ABB RobotStudio station: Tp2_20201215-221945.rsstn

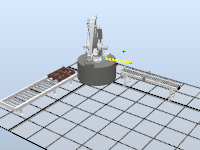
Station Tp2 (saved by RobotStudio 20.2.9116.0)
Controller Controlador1
  mechanical unit ROB_1: IRB660_180_315__01_2, 6 joints, base frame (0, 0, 1000) mm
Layout (positions relative to the parent item):
  - transporteCajas [part, from Equipment\Conveyor Guide 400.rslib] at (0, 1500, 0) mm, rotated rx 0 ry 0 rz 90 deg
  - Euro Pallet [graphiccomponentgroup, from Equipment\Euro Pallet.rslib] at (1000, -1425, 435) mm
    - Body 1 [part, from Equipment\Euro Pallet.rslib]
  - transportePallets [part, from Equipment\Conveyor 950 4000 h2.rslib] at (1000, -1500, 0) mm
  - IRB660_180_315__01_2 [mechanism, from Robots\IRB660_180_315__01.rslib] at (0, 0, 1000) mm; joint values [0.4389, 0.3282, 0.9586, 1.2589] (rad or m)
  - ventosa_tool [mechanism] at (1582.67, 743.05, 1659.86) mm, rotated rx 180 ry 0 rz 133.02 deg
      TCP ventosa_tool at (0, 0, 200) mm
      links: ventosa
  - pedestal [part]
  - fuenteBloques [smart component] at (-200, 1500, 770) mm
      signals: DI agarrar, DO cajaLista
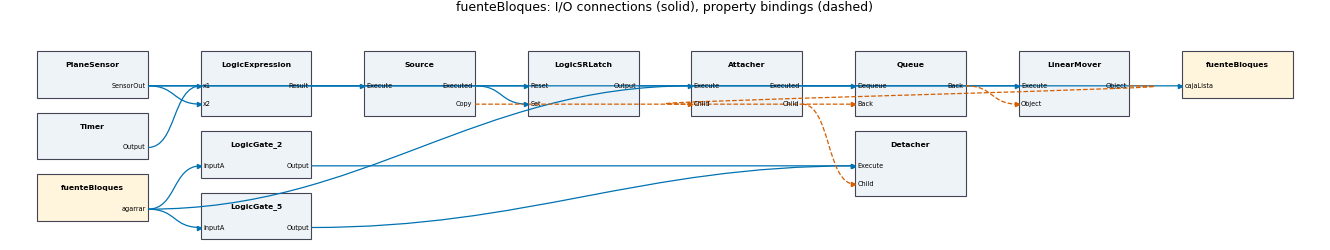
      connections:
        LogicSRLatch.Output -> LinearMover.Execute
        PlaneSensor.SensorOut -> LogicSRLatch.Reset
        Timer.Output -> LogicExpression.x1
        PlaneSensor.SensorOut -> LogicExpression.x2
        LogicExpression.Result -> Source.Execute
        Source.Executed -> LogicSRLatch.Set
        LogicGate_2.Output -> Detacher.Execute
        fuenteBloques.agarrar -> Attacher.Execute
        fuenteBloques.agarrar -> LogicGate_2.InputA
        PlaneSensor.SensorOut -> fuenteBloques.cajaLista
        Attacher.Executed -> Queue.Dequeue
        LogicGate_5.Output -> Detacher.Execute
        fuenteBloques.agarrar -> LogicGate_5.InputA
        Queue.Back => LinearMover.Object
        Source.Copy => Queue.Back
        LinearMover.Object => Attacher.Child
        Attacher.Child => Detacher.Child
    - Source [smart component, from Components\Source.rslib]
        properties: Source=caja; Copy=(none); Parent=(none); Position=[0 2.5 0]; Orientation=[0 0 0]; Transient=true; PhysicsBehavior=0
    - Timer [smart component, from Components\Timer.rslib]
        properties: StartTime=0; Interval=5; Repeat=true; CurrentTime=38.328
    - LinearMover [smart component, from Components\LinearMover.rslib]
        properties: Object=(none); Direction=[0 2.5 0]; Speed=-0.8; Reference=Local; ReferenceObject=fuenteBloques
    - PlaneSensor [smart component, from Components\PlaneSensor.rslib]
        properties: Origin=[-0.1 0.00100000000000011 0]; Axis1=[0 0 0.2]; Axis2=[0.2 0 0]; SensedPart=(none)
      - _sensorPart_ [part]
    - Queue [smart component, from Components\Queue.rslib]
        properties: Back=(none); Front=(none); Queue={b09acd23-45e5-4a9e-9d6f-6607265ff7c3};{23adc33f-3970-47e8-9e1c-f26a8dcf2bdc};{0d33cf10-6771-4310-8fb9-7d79b60af7e9};{83ef1169-329e-4ff4-9302-6302975186d9};{5ada7f3c-b0af-4a10-911f-6c2619dd6db8};{32b629fe-78aa-4961-aeab-383a7d5acd1b};{d9da9d26-80fb-4a26-bfbf-3b7bce0f61f2};{004fb7e2-83f2-4b9c-9668-500ebdcf4198};{63642d38-358b-4db6-ae17-5b4735758ac7};{fa627562-ab66-4e6f-ae79-46c97ebec96c};{c4f368e0-0d9a-4f43-8682-49ac6b133d0c};{43fd2dfd-2b72-4e17-8785-66f02cec94a6};{360d026e-603c-48f5-a2c0-6adaf5a54dd8};{faa924fc-b9a8-4cba-b3be-a1ab497ef86c};{72ea9125-d9f7-4887-b297-381c21b0fe64};{75f844bc-79ed-41e2-8179-ecb24b3a711f};{b9ae99bd-1fa5-4485-ae31-d081ce819117};{bdc3d345-f343-47d8-ada2-183b74e07857};{f98fed9e-0c76-4123-ac69-ce9101c203d3};{b8a068de-0981-4d01-b020-79f46d4aa61e};{6264e575-37ac-44c5-a35d-08152de0ecc4};{b9b05183-98bc-44b7-a44f-bd382026ea01};{e5950468-f040-4ced-9b2d-1f0ddcc9779f};{6daa5a7e-70c7-4fac-8eb8-a3f139030eec};{8209126b-952b-4f15-910a-db478de95a8e};{d94d3c0f-845f-4a91-8578-673738cefad5};{24218f6e-c39a-41e5-a039-2996c01a528f};{42922201-3d4c-4c3c-953c-a9a2c1819590};{11ce3d81-70fa-4fc5-817a-ad43dfd073f9};{d61a1e4e-17c4-421e-8ebd-c30096442b35};{77fdfff2-3eeb-40ed-8391-02d9a381d090};{a548ec3f-cf89-447b-a6c2-8c75641f384b};{21203246-2e5c-4335-a9cf-3c7fcd6009a5};{d9f34a10-d6ad-42c0-8e94-537fdd9e4098};{7434c9e7-4537-4421-8e6c-89bc8283500f};{b2407604-a6d2-40e8-b86b-a185e6f9dabb};{cfdb3468-085d-4a52-9af9-b93c9a7d77cb};{67c8250b-e61e-4164-96c4-8534bc7f99f1};{f8f70fdc-2725-4632-89b5-dc566ac6d74b};{9039b24f-4283-43ad-8f64-d17edb5e158d};{16ad2cc8-d29d-4a04-b806-8d5c79e89c70};{98e4d611-1296-4b4a-afc7-87a9f4683c65};{ea268e05-d762-4d6c-aedb-f9d60f45238b};{23698e1b-885b-404a-990f-58416227340d};{20caccea-1c23-41cc-8a6c-5124b1a7f711}; NumberOfObjects=1
    - caja [part]
    - LogicSRLatch [smart component, from Components\LogicSRLatch.rslib]
    - LogicExpression [smart component, from Components\LogicExpression.rslib]
        properties: Expression=x1 AND NOT x2
    - Attacher [smart component, from Components\Attacher.rslib]
        properties: Parent=ventosa_tool; Flange=0; Child=(none); Mount=false; Offset=[0 0 0]; Orientation=[0 0 0]
    - Detacher [smart component, from Components\Detacher.rslib]
        properties: Child=(none); KeepPosition=true
    - LogicGate_5 [smart component, from Components\LogicGate.rslib]
        properties: Operator=NOT; Delay=0
Attachment: Euro Pallet is attached to transportePallets
Attachment: ventosa_tool is attached to IRB660_180_315__01_2 / Link6
Attachment: pistaCajas is attached to transporteCajas
Attachment: pistaPallets is attached to transportePallets
Station logic (signal -> signal, property => property):
  Controlador1.do_pick -> fuenteBloques.agarrar
  fuenteBloques.cajaLista -> Controlador1.cajaLista
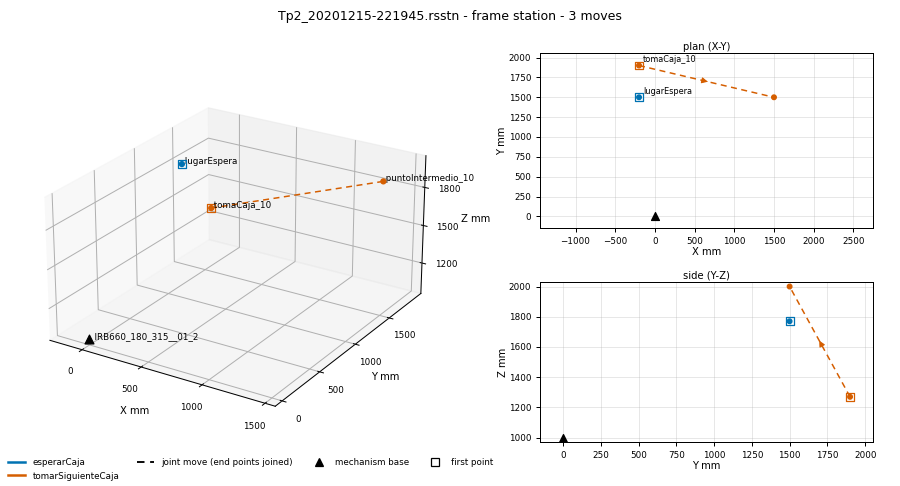
[picture p0: tool path of Tp2_20201215-221945.rsstn in frame station, 3 of 3 moves have a stored position in this frame; points joined in program order, loops and branches not executed]
Targets, tools, work objects and paths stored in the station, written as RAPID:
! task T_ROB1
MODULE Module1
  PERS tooldata ventosa_tool:=[TRUE,[[0,0,200],[1,0,0,0]],[1,[0,0,1],[1,0,0,0],0,0,0]];
  PERS wobjdata pistaCajas:=[FALSE,TRUE,"",[[-200,1500,770],[0,0,1,0]],[[0,0,0],[1,0,0,0]]];
  PERS wobjdata pistaPallets:=[FALSE,TRUE,"",[[1000,-1425,579],[0,0,1,0]],[[0,0,0],[1,0,0,0]]];
  CONST robtarget lugarEspera:=[[0,0,-1000],[1,0,0,0],[0,0,0,0],[9E+09,9E+09,9E+09,9E+09,9E+09,9E+09]];
  CONST robtarget tomaCaja_10:=[[0,400,-500],[1,0,0,0],[0,0,0,0],[9E+09,9E+09,9E+09,9E+09,9E+09,9E+09]];
  CONST robtarget superficiePallet_10:=[[0,0,0],[1,0,0,0],[0,0,0,0],[9E+09,9E+09,9E+09,9E+09,9E+09,9E+09]];
  CONST robtarget puntoIntermedio_10:=[[1500,1500,2000],[0,0,1,0],[0,0,0,0],[9E+09,9E+09,9E+09,9E+09,9E+09,9E+09]];
  PROC main()
    SetDO do_pick,0;
    esperarCaja;
    tomarSiguienteCaja;
    esperarCaja;
  ENDPROC
  PROC esperarCaja()
    MoveJ lugarEspera,v1000,fine,ventosa_tool\WObj:=pistaCajas;
    WaitDI cajaLista,1;
  ENDPROC
  PROC tomarSiguienteCaja()
    MoveJ tomaCaja_10,v1000,fine,ventosa_tool\WObj:=pistaCajas;
    SetDO do_pick,1;
    MoveJ puntoIntermedio_10,v1000,z100,ventosa_tool\WObj:=wobj0;
  ENDPROC
ENDMODULE

